// TwinCAT 3 PLC project LiquidTank
// ProgramVersion: 3.1.4024.0
// libraries:
//   Tc2_Standard, * (Beckhoff Automation GmbH)
//   Tc2_System, * (Beckhoff Automation GmbH)
//   Tc3_Module, * (Beckhoff Automation GmbH)
// project tree:
//   / GlobalTextList.TcGTLO, PlcTask.TcTTO, Visualization Manager.TcVMO (not stored)
//   POUs/ FB_BlinkingLight.TcPOU, FB_Button.TcPOU, FB_ButtonT.TcPOU, FB_Tank.TcPOU, MAIN.TcPOU
//   VISUs/ Visualization.TcVIS

CONFIGURATION LiquidTank
    RESOURCE PLC ON TwinCAT3
        TASK PlcTask(INTERVAL := T#10ms, PRIORITY := 20);
        PROGRAM MAIN WITH PlcTask : MAIN;
    END_RESOURCE
END_CONFIGURATION

// ---- POUs/MAIN.TcPOU
PROGRAM MAIN
VAR
	fbLiquidTank : FB_Tank; 	

	bFillButton : BOOL;
	bDrainButton : BOOL;
END_VAR

fbLiquidTank(bIsFillButtonPressed := bFillButton, bIsDrainButtonPressed := bDrainButton);

END_PROGRAM

// ---- POUs/FB_Tank.TcPOU
FUNCTION_BLOCK FB_Tank
VAR_INPUT
	bIsFillButtonPressed : BOOL;
	bIsDrainButtonPressed : BOOL;
END_VAR
VAR_OUTPUT
	bFillValve : BOOL;
	bDrainValve : BOOL;
	
	bFillLight : BOOL;
	bDrainLight : BOOL;
	
	bFillBlink : BOOL;
	bDrainBlink : BOOL;
END_VAR
VAR
	// Instances of the button FB
	fbFillButton : FB_Button;
	fbDrainButton : FB_Button;
	
	fbFButton : FB_ButtonT;
	fbDButton : FB_ButtonT;

	fbFillLightBlink : FB_BlinkingLight;
	fbDrainLightBlink : FB_BlinkingLight;

	CurrentState : INT;
	
	// bIsFilling : BOOL;
	// bIsDraining : BOOL;
	
	fbFillTimer : TON;
	fbDrainTimer : TON;
	
	tMaxTime : TIME := T#6S;	// Maximum time it takes the tank to fill / drain
	tFillTime : TIME := tMaxTime;	// Remaining time it takes to fill the tank
	tDrainTime : TIME := tMaxTime;	// Remaining time it takes to drain the tank
	
	tElapsedFillTime : TIME;
	tElapsedDrainTime : TIME;
	
	bHighSensor : BOOL;
	bLowSensor : BOOL;
	
	fbFillStop : R_TRIG;
	fbDrainStop : R_TRIG;
	
	// Variables used only for the visualisation
	bVisHigh : BOOL;
	bVisMid : BOOL;
	bVisLow : BOOL;
	fbVisTimer1 : TON;
	fbVisTimer2 : TON;
	
	Pomoshen : TON;
	bPom : BOOL;
	
	bProcessStopped: BOOL;
	bAllowFilling: BOOL := TRUE;
	
	bActivate : BOOL;
END_VAR

// State machine logic
CASE currentState OF
    0: // Idle
        bFillValve := FALSE;
        bDrainValve := FALSE;

        bFillLight := FALSE;
        bDrainLight := FALSE;

        bFillBlink := FALSE;
        bDrainBlink := FALSE;

        fbFillTimer.IN := FALSE;
        fbDrainTimer.IN := FALSE;

        IF fbFillButton.bActivate AND NOT bHighSensor THEN
            currentState := 1; // Filling
        ELSIF fbDrainButton.bActivate AND NOT bLowSensor THEN
            currentState := 2; // Draining
        END_IF

    1: // Filling
        bFillValve := TRUE;
        bDrainValve := FALSE;

        fbFillLightBlink(dwTimeOn := 500, dwTimeOff := 250, bLight => bFillLight);
        bDrainLight := FALSE;

        fbFillTimer.IN := TRUE;
        fbDrainTimer.IN := FALSE;

        tElapsedFillTime := fbFillTimer.ET;
		
		fbVisTimer1(IN := TRUE);
		IF fbVisTimer1.Q THEN
			bVisHigh := FALSE;
			bVisMid := FALSE;
			bVisLow := TRUE;
		END_IF
		fbVisTimer2(IN := TRUE);
		IF fbVisTimer2.Q THEN
			bVisHigh := FALSE;
			bVisMid := TRUE;
			bVisLow := TRUE;
		END_IF

        IF bHighSensor THEN
            bLowSensor := FALSE;
			
			fbVisTimer1(IN := FALSE);
			fbVisTimer2(IN := FALSE);
			
			bVisHigh := TRUE;
			bVisMid := TRUE;
			bVisLow := TRUE;
			
            currentState := 3; // Full
        END_IF

    2: // Draining
        bFillValve := FALSE;
        bDrainValve := TRUE;

        bFillLight := FALSE;
        fbDrainLightBlink(dwTimeOn := 500, dwTimeOff := 250, bLight => bDrainLight);

        fbFillTimer.IN := FALSE;
        fbDrainTimer.IN := TRUE;

        tElapsedDrainTime := fbDrainTimer.ET;
		
		fbVisTimer1(IN := TRUE);
		IF fbVisTimer1.Q THEN
			bVisHigh := FALSE;
			bVisMid := TRUE;
			bVisLow := TRUE;
		END_IF
		fbVisTimer2(IN := TRUE);
		IF fbVisTimer2.Q THEN
			bVisHigh := FALSE;
			bVisMid := FALSE;
			bVisLow := TRUE;
		END_IF

        IF bLowSensor THEN
            bHighSensor := FALSE;
			
			fbVisTimer1(IN := FALSE);
			fbVisTimer2(IN := FALSE);
			
			bVisHigh := FALSE;
			bVisMid := FALSE;
			bVisLow := FALSE;
			
            currentState := 4; // Empty
        END_IF

    3: // Full
        bFillValve := FALSE;
        bFillLight := TRUE;

        bHighSensor := TRUE;
        bLowSensor := FALSE;

        bDrainValve := FALSE;

        IF fbDrainButton.bActivate THEN
            fbDrainTimer.IN := TRUE;
            fbFillTimer.IN := FALSE;
            currentState := 2; // Draining
        END_IF

    4: // Empty
        bDrainValve := FALSE;
        bDrainLight := TRUE;

        bHighSensor := FALSE;
        bLowSensor := TRUE;

        IF fbFillButton.bActivate THEN
            currentState := 1; // Filling
        END_IF
END_CASE

// Update button states
fbFillButton(bIsButtonPressed := bIsFillButtonPressed);
fbDrainButton(bIsButtonPressed := bIsDrainButtonPressed);

// Update timers based on button deactivation and state changes
IF (NOT fbFillButton.bActivate AND currentState = 1) THEN
    tFillTime := tMaxTime - tElapsedFillTime;
    tDrainTime := tElapsedFillTime;	
    currentState := 0; // Transition to Idle
ELSIF (NOT fbDrainButton.bActivate AND currentState = 2) THEN
    tDrainTime := tMaxTime - tElapsedDrainTime;
    tFillTime := tElapsedDrainTime;
    currentState := 0; // Transition to Idle
ELSIF (NOT fbFillButton.bActivate AND currentState = 3) THEN
    tFillTime := T#0S;
    tDrainTime := tMaxTime;	
    currentState := 0; // Transition to Idle
ELSIF (NOT fbDrainButton.bActivate AND currentState = 4) THEN
    tFillTime := tMaxTime;
    tDrainTime := T#0S;	
    currentState := 0; // Transition to Idle
END_IF

// Sensor logic
IF bFillValve THEN
    tElapsedFillTime := fbFillTimer.ET;
    IF fbFillTimer.Q THEN
        bHighSensor := TRUE;
        bLowSensor := FALSE;
    ELSE
        bHighSensor := FALSE;
        bLowSensor := FALSE;
    END_IF
END_IF

IF bDrainValve THEN
    tElapsedDrainTime := fbDrainTimer.ET;
    IF fbDrainTimer.Q THEN
        bHighSensor := FALSE;
        bLowSensor := TRUE;
    ELSE
        bHighSensor := FALSE;
        bLowSensor := FALSE;
    END_IF
END_IF

fbFillTimer(PT := tFillTime);
fbDrainTimer(PT := tDrainTime);

fbVisTimer1(PT := T#2S);
fbVisTimer2(PT := T#4S);














//// State machine logic
//CASE currentState OF
//    0: // Idle
//        bFillValve := FALSE;
//        bDrainValve := FALSE;

//        bFillLight := FALSE;
//        bDrainLight := FALSE;

//        bFillBlink := FALSE;
//        bDrainBlink := FALSE;

//        fbFillTimer.IN := FALSE;
//        fbDrainTimer.IN := FALSE;

//        IF fbFButton.bActivate AND NOT bHighSensor THEN
//            currentState := 1; // Filling
//        ELSIF fbDButton.bActivate AND NOT bLowSensor THEN
//            currentState := 2; // Draining
//        END_IF

//    1: // Filling
//        bFillValve := TRUE;
//        bDrainValve := FALSE;

//        fbFillLightBlink(dwTimeOn := 500, dwTimeOff := 250, bLight => bFillLight);
//        bDrainLight := FALSE;

//        fbFillTimer.IN := TRUE;
//        fbDrainTimer.IN := FALSE;

//        tElapsedFillTime := fbFillTimer.ET;
		
//		fbVisTimer1(IN := TRUE);
//		IF fbVisTimer1.Q THEN
//			bVisHigh := FALSE;
//			bVisMid := FALSE;
//			bVisLow := TRUE;
//		END_IF
//		fbVisTimer2(IN := TRUE);
//		IF fbVisTimer2.Q THEN
//			bVisHigh := FALSE;
//			bVisMid := TRUE;
//			bVisLow := TRUE;
//		END_IF

//        IF bHighSensor THEN
//            bLowSensor := FALSE;
			
//			fbVisTimer1(IN := FALSE);
//			fbVisTimer2(IN := FALSE);
			
//			bVisHigh := TRUE;
//			bVisMid := TRUE;
//			bVisLow := TRUE;
			
//            currentState := 3; // Full
//        END_IF

//    2: // Draining
//        bFillValve := FALSE;
//        bDrainValve := TRUE;

//        bFillLight := FALSE;
//        fbDrainLightBlink(dwTimeOn := 500, dwTimeOff := 250, bLight => bDrainLight);

//        fbFillTimer.IN := FALSE;
//        fbDrainTimer.IN := TRUE;

//        tElapsedDrainTime := fbDrainTimer.ET;
		
//		fbVisTimer1(IN := TRUE);
//		IF fbVisTimer1.Q THEN
//			bVisHigh := FALSE;
//			bVisMid := TRUE;
//			bVisLow := TRUE;
//		END_IF
//		fbVisTimer2(IN := TRUE);
//		IF fbVisTimer2.Q THEN
//			bVisHigh := FALSE;
//			bVisMid := FALSE;
//			bVisLow := TRUE;
//		END_IF

//        IF bLowSensor THEN
//            bHighSensor := FALSE;
			
//			fbVisTimer1(IN := FALSE);
//			fbVisTimer2(IN := FALSE);
			
//			bVisHigh := FALSE;
//			bVisMid := FALSE;
//			bVisLow := FALSE;
			
//            currentState := 4; // Empty
//        END_IF

//    3: // Full
//        bFillValve := FALSE;
//        bFillLight := TRUE;

//        bHighSensor := TRUE;
//        bLowSensor := FALSE;

//        bDrainValve := FALSE;

//        IF fbDButton.bActivate THEN
//            fbDrainTimer.IN := TRUE;
//            fbFillTimer.IN := FALSE;
//            currentState := 2; // Draining
//        END_IF

//    4: // Empty
//        bDrainValve := FALSE;
//        bDrainLight := TRUE;

//        bHighSensor := FALSE;
//        bLowSensor := TRUE;

//        IF fbFButton.bActivate THEN
//            currentState := 1; // Filling
//        END_IF
//END_CASE

//// Update button states
//fbFButton(bIsButtonOn := bIsFillButtonPressed);
//fbDButton(bIsButtonOn := bIsDrainButtonPressed);

////// Update timers based on button deactivation and state changes
////IF (NOT fbFButton.bActivate AND currentState = 1) THEN
////    tFillTime := tMaxTime - tElapsedFillTime;
////    tDrainTime := tElapsedFillTime;	
////    currentState := 0; // Transition to Idle
////ELSIF (NOT fbDButton.bActivate AND currentState = 2) THEN
////    tDrainTime := tMaxTime - tElapsedDrainTime;
////    tFillTime := tElapsedDrainTime;
////    currentState := 0; // Transition to Idle
////ELSIF (NOT fbFButton.bActivate AND currentState = 3) THEN
////    tFillTime := T#0S;
////    tDrainTime := tMaxTime;	
////    currentState := 0; // Transition to Idle
////ELSIF (NOT fbDButton.bActivate AND currentState = 4) THEN
////    tFillTime := tMaxTime;
////    tDrainTime := T#0S;	
////    currentState := 0; // Transition to Idle
////END_IF

//IF (NOT fbFButton.bActivate AND currentState = 1) THEN
//    tFillTime := tMaxTime - tElapsedFillTime;
//    tDrainTime := tElapsedFillTime;	
//    currentState := 0; // Transition to Idle
//ELSIF (NOT fbDButton.bActivate AND currentState = 2) THEN
//    tDrainTime := tMaxTime - tElapsedDrainTime;
//    tFillTime := tElapsedDrainTime;
//    currentState := 0; // Transition to Idle
//ELSIF (NOT fbFButton.bActivate AND currentState = 3) THEN
//    tFillTime := T#0S;
//    tDrainTime := tMaxTime;	
//    currentState := 0; // Transition to Idle
//ELSIF (NOT fbDButton.bActivate AND currentState = 4) THEN
//    tFillTime := tMaxTime;
//    tDrainTime := T#0S;	
//    currentState := 0; // Transition to Idle
//END_IF


//// Sensor logic
//IF bFillValve THEN
//    tElapsedFillTime := fbFillTimer.ET;
//    IF fbFillTimer.Q THEN
//        bHighSensor := TRUE;
//        bLowSensor := FALSE;
		
//		fbFButton(bIsButtonOff := TRUE);
//    ELSE
//        bHighSensor := FALSE;
//        bLowSensor := FALSE;
//    END_IF
//END_IF

//IF bDrainValve THEN
//    tElapsedDrainTime := fbDrainTimer.ET;
//    IF fbDrainTimer.Q THEN
//        bHighSensor := FALSE;
//        bLowSensor := TRUE;
		
//		fbDButton(bIsButtonOff := TRUE);
//    ELSE
//        bHighSensor := FALSE;
//        bLowSensor := FALSE;
//    END_IF
//END_IF

//fbFillTimer(PT := tFillTime);
//fbDrainTimer(PT := tDrainTime);

//fbVisTimer1(PT := T#2S);
//fbVisTimer2(PT := T#4S);

END_FUNCTION_BLOCK

// ---- POUs/FB_Button.TcPOU
FUNCTION_BLOCK FB_Button
VAR_INPUT
	bIsButtonPressed : BOOL;
END_VAR
VAR_OUTPUT
	bActivate : BOOL;
END_VAR
VAR
	fbToggle_RTRIG : R_TRIG;
END_VAR

// This is a toggle button
fbToggle_RTRIG(clk := bIsButtonPressed);
IF fbToggle_RTRIG.Q THEN
	bActivate := NOT bActivate;
END_IF

END_FUNCTION_BLOCK

// ---- POUs/FB_ButtonT.TcPOU
FUNCTION_BLOCK FB_ButtonT
VAR_INPUT
	bIsButtonOn : BOOL;
	bIsButtonOff : BOOL;
END_VAR
VAR_OUTPUT
	bActivate : BOOL;
END_VAR
VAR
	fbOn_RTRIG : R_TRIG;
	fbOff_RTRIG : R_TRIG;
END_VAR

// One button turns the light on, the other turns it off
IF bIsButtonOn THEN
	bActivate := TRUE;
	bIsButtonOff := FALSE;
END_IF

IF bIsButtonOff THEN
	bActivate := FALSE;
	bIsButtonOn := FALSE;
END_IF

END_FUNCTION_BLOCK

// ---- POUs/FB_BlinkingLight.TcPOU
FUNCTION_BLOCK FB_BlinkingLight
VAR_INPUT
	dwTimeOn : DWORD;
	dwTimeOff : DWORD;
END_VAR
VAR_OUTPUT
	bLight : BOOL;	// Determines whether the light will be ON or OFF
END_VAR
VAR
	fbTimerOn : TON;
	fbTimerOff : TON;
	fbStartTrigger : R_TRIG;
	
	nCurrentPhase : INT := 10;	// 10 - ON, 20 - OFF
	
	bIsBlinking : bool;
END_VAR

CASE nCurrentPhase OF
    10:	// ON
        fbTimerOn(IN := TRUE, PT := DWORD_TO_TIME(dwTimeOn));
        IF fbTimerOn.Q THEN
            fbTimerOn(IN := FALSE); // Reset the on timer
            nCurrentPhase := 20;  // Move to the off phase
        END_IF
        bLight := TRUE;

    20:	// OFF
        fbTimerOff(IN := TRUE, PT := DWORD_TO_TIME(dwTimeOff));
        IF fbTimerOff.Q THEN
            fbTimerOff(IN := FALSE); // Reset the off timer
            nCurrentPhase := 10;  // Move to the On phase
        END_IF
        bLight := FALSE;
		
ELSE
	fbTimerOn(IN := FALSE);
    fbTimerOff(IN := FALSE);
    bLight := FALSE;
END_CASE

END_FUNCTION_BLOCK

// ---- GlobalTextList.TcGTLO
TEXTLIST GlobalTextList
  997 = 'Drain'
  965 = 'Fill'
  50 = 'Tank'
END_TEXTLIST

// ---- VISUs/Visualization.TcVIS
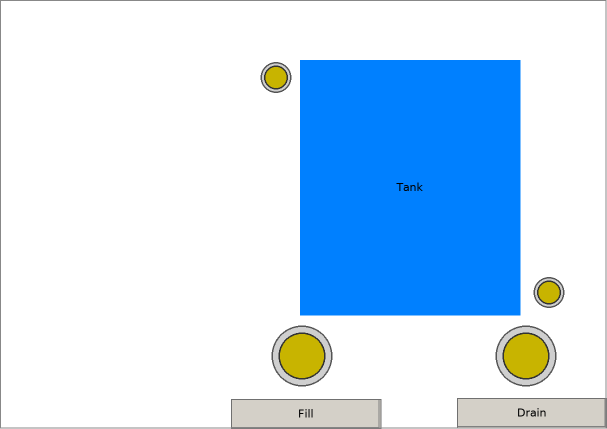
VISUALIZATION Visualization  // 607x429
    Lamp1 (267,321 70x70), variable: MAIN.fbLiquidTank.bFillLight, style: Lamp-Lamp1-Yellow
    Lamp1 (491,321 70x70), variable: MAIN.fbLiquidTank.bDrainLight, style: Lamp-Lamp1-Yellow
    Button (231,399 150x30), "Fill"
        tap MAIN.bFillButton
    Button (457,398 150x30), "Drain"
        tap MAIN.bDrainButton
    Rectangle (300,60 220x255), "Tank"
    Rectangle (300,145 220x85), "Tank", invisible if: NOT MAIN.fbLiquidTank.bVisMid
    Rectangle (300,60 220x85), invisible if: NOT MAIN.fbLiquidTank.bVisHigh
    Rectangle (300,230 220x85), invisible if: NOT MAIN.fbLiquidTank.bVisLow
    Lamp1 (258,58 36x39), variable: MAIN.fbLiquidTank.bHighSensor, style: Lamp-Lamp1-Yellow
    Lamp1 (531,273 36x39), variable: MAIN.fbLiquidTank.bLowSensor, style: Lamp-Lamp1-Yellow
END_VISUALIZATION
